RoboDK station: CuadrosElectricos.rdk

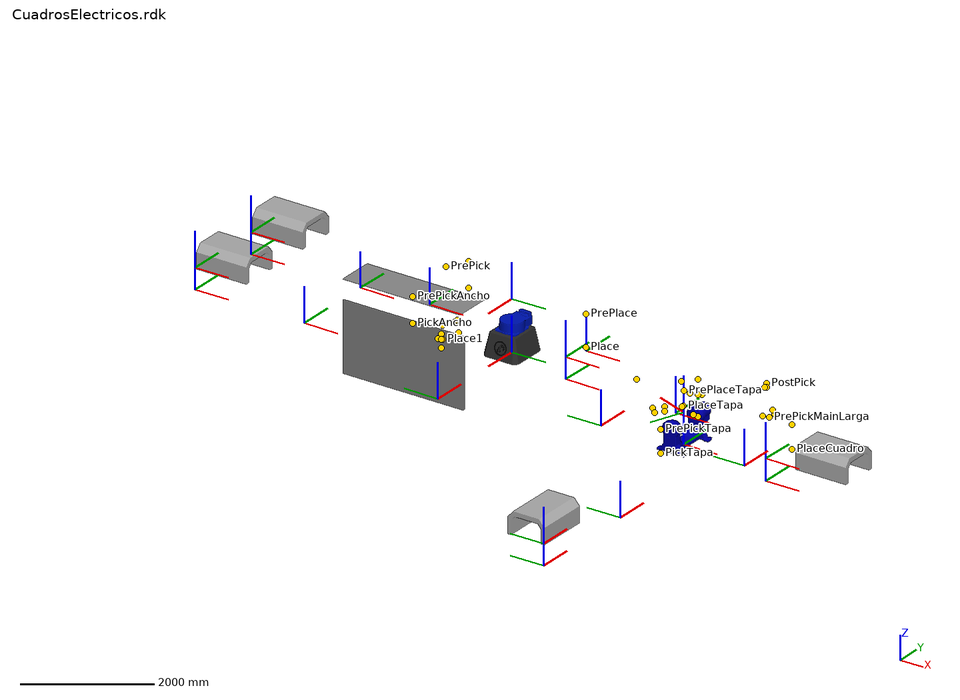
[picture v0: the station drawn from its stored meshes, robots at their saved joint values, targets as dots, program paths as lines]
Station CuadrosElectricos (saved by RoboDK 6.0.0). Poses are relative to the parent item; angles as X-Y-Z fixed-axis rotations.
Station parameters (name, value as stored): SensorCA, 0, SensorCL, 0, SensorCM, 0, SensorTapa, 0, SensorEtiqueta, 0, SensorFinalEtiqueta, 0, BendingHecho, 0, enCintaMain, 0, mesaOcupada, 0, LasDos, 0, planchaSoldada, 0, tapaPuesta, 0, EnCintaEtiquetar, 0, numero_planchaAncha, 0, numero_planchaLarga, 0, numero_planchaAncha1, 0, numero_planchaAncha2, 0, numero_planchaLarga1, 0, numero_planchaLarga2, 0, numero_planchaSoldada, 0, numero_tapaCuadro, 0, numero_cuadroConTapa, 0, numero_cuadroEtiquetada, 0, yaskawa_larga, 0, yaskawa_ancha, 0, abb_tapa, 0, parada_emergencia, 0
  - machining project Ajustes de mecanizado1: rotZ(0) | rotX(0)*rotY(0) | rotz(0) | onStart | onPathStart | onApproach | onPoint | onRetract | onFinish | SetRPM(%1) | SetTool(%1) | Extruder(%1) | default | default | OutOnMov(%1) | OutOffMov(%1) | onPathFinish | M_RunCode(%1)
  - folder Sistemas de Ref
    - frame World at (0, 0, 0) mm, rotated rx 0 ry 0 rz -90 deg
      - object Valla at (10, -2980, 0) mm, rotated rx 0 ry 0 rz 90 deg
      - object PedestalRobotPrensado at (0, 0, 0) mm, rotated rx 0 ry 0 rz 90 deg, size 633.4 x 700.2 x 375 mm, 1065353216 curves, geometry from Pedestal-H500mm-Type-2 (1).sld
      - object Suelo at (1170, 1000, -5) mm, size 11520 x 17280 x 0 mm, 1056816382 curves, geometry from PLUGIN_DISPLAY_DATAU
      - frame Frame_CintaCuadroInit at (300, 1190, 0) mm, rotated rx 0 ry 0 rz 90 deg
        - robot CintaCuadroIni: 1 axes
            modified DH rows (alpha deg, a mm, theta deg, d mm): 0, 0, 0, 0 linear
            base shift (0, 0, 0) mm, rotated rx 0 ry 90 rz 0 deg
            joint limits [-900000] to [900000]; home [0]; saved at [0]
          - frame FramePlanchaMain at (0, 0, 0) mm
      - frame Frame_CintaCuadroMid at (300, 3190, 0) mm, rotated rx 0 ry 0 rz 90 deg
        - robot CintaCuadroMid: 1 axes
            modified DH rows (alpha deg, a mm, theta deg, d mm): 0, 0, 0, 0 linear
            base shift (0, 0, 0) mm, rotated rx 0 ry 90 rz 0 deg
            joint limits [-900000] to [900000]; home [0]; saved at [0]
        - object SensorCM at (1880, 630, 370) mm, rotated rx 90 ry 0 rz -90 deg
      - frame Frame_CintaCuadroFinal at (1420, 5610, 0) mm, rotated rx 0 ry 0 rz 90 deg
        - robot CintaCuadroFini: 1 axes
            modified DH rows (alpha deg, a mm, theta deg, d mm): 0, 0, 0, 0 linear
            base shift (0, 0, 0) mm, rotated rx 0 ry 90 rz 0 deg
            joint limits [-900000] to [900000]; home [0]; saved at [0]
          - frame FrameEtiqueta at (0, 0, 0) mm
        - target CintaCuadroSoldadoIni (joint target) at (-550, 0, 366.5) mm; joints [3450] of CintaCuadroFini
        - target CintaCuadroSoldadoFin (joint target) at (2010, 0, 366.5) mm; joints [6010, -103.845, 100.785, 0, -114.63, -14.149, 0] of CintaCuadroFini
        - object tunelEtiqueta at (1000, 310, 760) mm, size 913.4 x 675.6 x 396.2 mm, geometry from tunel_andreu.stl
        - object SensorEtiqueta at (1240, 310, 690) mm, rotated rx 0 ry 90 rz 0 deg
        - object SensorFinalEtiqueta at (1880, 630, 370) mm, rotated rx 90 ry 0 rz -90 deg
      - frame Frame_CintaAnchoInit at (970, -5100, 0) mm, rotated rx 0 ry 0 rz 90 deg
        - robot CintaAnchoIni: 1 axes
            modified DH rows (alpha deg, a mm, theta deg, d mm): 0, 0, 0, 0 linear
            base shift (0, 0, 0) mm, rotated rx 0 ry 90 rz 0 deg
            joint limits [-900000] to [900000]; home [0]; saved at [0]
          - frame FramePlanchaAncha at (9, 0, 0) mm
        - object tunelAncha at (-2360, 3530, -20) mm, size 913.4 x 675.6 x 396.2 mm, geometry from tunel_andreu.stl
      - frame Frame_CintaAnchoFinal at (970, -3100, 0) mm, rotated rx 0 ry 0 rz 90 deg
        - robot Conveyor Belt Wide (2m): 1 axes
            modified DH rows (alpha deg, a mm, theta deg, d mm): 0, 0, 0, 0 linear
            base shift (0, 0, 0) mm, rotated rx 0 ry 90 rz 0 deg
            joint limits [-900000] to [900000]; home [0]; saved at [28.931]
        - object SensorCA at (1915, -40, 351.5) mm, rotated rx 90 ry 0 rz 90 deg
      - frame Frame_CintaLargoInit at (-490, -5100, 0) mm, rotated rx 0 ry 0 rz 90 deg
        - robot CintaLargoIni: 1 axes
            modified DH rows (alpha deg, a mm, theta deg, d mm): 0, 0, 0, 0 linear
            base shift (0, 0, 0) mm, rotated rx 0 ry 90 rz 0 deg
            joint limits [-900000] to [900000]; home [0]; saved at [0]
          - frame FramePlanchaLarga at (0, 0, 0) mm
        - object tunelLarga at (-2360, 3530, -20) mm, size 913.4 x 675.6 x 396.2 mm, geometry from tunel_andreu.stl
      - frame Frame_CintaLargoFinal at (-490, -3100, 0) mm, rotated rx 0 ry 0 rz 90 deg
        - robot Conveyor Belt Wide (2m): 1 axes
            modified DH rows (alpha deg, a mm, theta deg, d mm): 0, 0, 0, 0 linear
            base shift (0, 0, 0) mm, rotated rx 0 ry 90 rz 0 deg
            joint limits [-900000] to [900000]; home [0]; saved at [28.931]
        - object SensorCL at (1825, -40, 351.5) mm, rotated rx 90 ry 0 rz 90 deg
      - frame Frame_CintaTapaInit at (5690, 4560, 0) mm, rotated rx 0 ry 0 rz 180 deg
        - robot CintaTapaInit: 1 axes
            modified DH rows (alpha deg, a mm, theta deg, d mm): 0, 0, 0, 0 linear
            base shift (0, 0, 0) mm, rotated rx 0 ry 90 rz 0 deg
            joint limits [-900000] to [900000]; home [0]; saved at [0]
          - frame FrameTapa at (0, 0, 0) mm
        - object tunelTapa at (-2430, 3530, -20) mm, size 913.4 x 675.6 x 396.2 mm, geometry from tunel_andreu.stl
      - frame Frame_CintaTapaFinal at (3690, 4560, 0) mm, rotated rx 0 ry 0 rz 180 deg
        - robot CintaTapaFinal: 1 axes
            modified DH rows (alpha deg, a mm, theta deg, d mm): 0, 0, 0, 0 linear
            base shift (0, 0, 0) mm, rotated rx 0 ry 90 rz 0 deg
            joint limits [-900000] to [900000]; home [0]; saved at [3450]
        - object SensorTapa at (1710, 620, 355) mm, rotated rx 90 ry 0 rz -90 deg
    - frame RobotPrensado at (0, 0, 880) mm, rotated rx 0 ry 0 rz -90 deg
      - robot Yaskawa MH24 Prensado (model Yaskawa MH24): 6 axes, payload 24 kg, reach 1730 mm, repeatability 0.06 mm, weight 268 kg
          modified DH rows (alpha deg, a mm, theta deg, d mm): 0, 0, 0, 505; -90, 150, -90, 0; 0, 760, 0, 0; -90, 200, 0, 795; 90, 0, 0, 0; -90, 0, 0, 100
          base shift (0, 0, -505) mm
          joint limits [-180, -105, -170, -200, -150, -455] to [180, 155, 240, 200, 150, 455]; home [0, 0, 0, 0, 0, 0]; saved at [-120.522, 54.399, 24.171, 0, -59.772, 120.522]
        - tool EPick Bend, TCP at (0, 0, 185) mm
    - frame RobotPaletizado at (5060, -1180, 0) mm, rotated rx 0 ry 0 rz 90 deg
      - robot ABB Paletizado (model ABB IRB 1660-4/1.55): 6 axes, payload 4 kg, reach 1550 mm, repeatability 0.02 mm, weight 257 kg
          modified DH rows (alpha deg, a mm, theta deg, d mm): 0, 0, 0, 481.5; -90, 150, -90, 0; 0, 700, 0, 0; -90, 110, 0, 678; 90, 0, 0, 0; -90, 0, 180, 135
          joint limits [-180, -90, -238, -175, -120, -400] to [180, 150, 79, 175, 120, 400]; home [0, 0, 0, 0, 0, 0]; saved at [16.288, 32.625, 48.175, 16.099, -82.213, 87.26]
        - tool EPick Gripper, TCP at (0, 30, 180) mm
      - frame Cinta_Mesa at (0, 0, 0) mm
        - target PrePickMainLarga (Cartesian target) at (777.3, 95, 463.61) mm, rotated rx 88.94 ry 0.2 rz 90.34 deg; joints [11.364, 25.315, 71.994, 11.14, -98.231, 91.211, 0] of ABB Paletizado
        - target PickMainLarga (Cartesian target) at (927.3, 95, 463.61) mm, rotated rx 88.94 ry 0.2 rz 90.33 deg; joints [8.631, 27.949, 59.348, 8.295, -88.383, 89.412, 0] of ABB Paletizado
        - target PrePickMainAncha (Cartesian target) at (777, 210.74, 455.18) mm, rotated rx 88.94 ry 0.2 rz 90.34 deg; joints [24.29, 27.02, 68.896, 24.11, -96.462, 92.216, 0] of ABB Paletizado
        - target PickMainAncha (Cartesian target) at (1028.89, 210.74, 455.18) mm, rotated rx 88.94 ry 0.2 rz 90.34 deg; joints [16.288, 32.625, 48.175, 16.099, -82.213, 87.26, 0] of ABB Paletizado
        - target PostPick (Cartesian target) at (758.49, 121.16, 1025.46) mm, rotated rx 88.94 ry 0.2 rz 90.34 deg; joints [15.024, -32.079, 48.401, 41.2, -22.631, 50.585, 0] of ABB Paletizado
        - target Giro180_P (Cartesian target) at (758, 121, 965.48) mm, rotated rx -88.95 ry -1.49 rz -89.69 deg; joints [15.162, -32.222, 48.464, 41.609, -22.656, 228.889, 0] of ABB Paletizado
        - target PrePlaceMain (Cartesian target) at (-1.33, 767.63, 965.52) mm, rotated rx -88.95 ry -1.51 rz -8.65 deg; joints [96.19, -32.22, 48.46, 41.6, -22.65, 228.88, 0] of ABB Paletizado
        - target PlaceMainLarga (Cartesian target) at (82, 907.5, 524) mm, rotated rx -90 ry 0 rz 0 deg; joints [82.121, 11.477, 61.016, -8.257, -72.663, -87.524, 0] of ABB Paletizado
        - target PlaceMainAncha (Cartesian target) at (100, 995, 525) mm, rotated rx -90 ry 0 rz 0 deg; joints [81.634, 16.501, 53.189, -8.912, -69.916, -86.918, 0] of ABB Paletizado
      - target Inicio (Cartesian target) at (790.15, 181.03, 936.03) mm, rotated rx 88.94 ry 0.2 rz 90.33 deg; joints [20.625, -24.78, 52.397, 37.542, -34.674, 57.118, 0] of ABB Paletizado
      - target PrePickTapa (Cartesian target) at (-1018.21, 818.52, 780.95) mm, rotated rx -179.33 ry -0.3 rz -86.99 deg; joints [140.371, 40.682, -38.487, -0.236, 88.496, 47.366, 0] of ABB Paletizado
      - target PickTapa (Cartesian target) at (-1018.21, 818.52, 380.95) mm, rotated rx -179.33 ry -0.3 rz -86.99 deg; joints [140.371, 46.29, -14.025, -0.277, 58.427, 47.505, 0] of ABB Paletizado
      - target PrePlaceTapa (Cartesian target) at (77.73, 1160.64, 889) mm, rotated rx -179.72 ry 0.67 rz -177.45 deg; joints [86.193, 25.731, -24.216, -0.695, 88.694, 83.664, 0] of ABB Paletizado
      - target PrePlaceTapaG1 (Cartesian target) at (239.54, 1017.6, 1052.03) mm, rotated rx 108.26 ry -87.33 rz -106.91 deg; joints [60.84, 25.81, -11.886, 81.018, 119.265, 70.969, 0] of ABB Paletizado
      - target PrePlaceTapaG2 (Cartesian target) at (239.54, 1017.6, 802.03) mm, rotated rx 108.26 ry -87.33 rz -106.91 deg; joints [60.84, 30.993, 1.938, 71.52, 114.698, 50.23, 0] of ABB Paletizado
      - target PrePlaceTapaG3 (Cartesian target) at (243.81, 1163, 773.67) mm, rotated rx 105.66 ry -86.91 rz -104.31 deg; joints [63.869, 42.236, -14.07, 75.44, 113.553, 55.604, 0] of ABB Paletizado
      - target PlaceTapa (Cartesian target) at (86.58, 1170.89, 626.96) mm, rotated rx -179.79 ry -0.03 rz -176.92 deg; joints [85.58, 27.86, -5.32, 0, 67.67, 82.5, 0] of ABB Paletizado
      - target PrePickCuadro (Cartesian target) at (51.62, 1181.79, 1052.12) mm, rotated rx -179.77 ry 0.7 rz 177.71 deg; joints [87.684, 33.633, -50.583, -0.729, 107.181, 89.762, 0] of ABB Paletizado
      - target PickCuadro (Cartesian target) at (56.65, 1179.89, 632.15) mm, rotated rx -179.77 ry 0.7 rz 177.71 deg; joints [87.43, 28.34, -6.48, -0.75, 68.37, 90, 0] of ABB Paletizado
      - target PrePlaceCuadro (Cartesian target) at (82.65, -808.13, 869.56) mm, rotated rx 179.56 ry -0.46 rz -2.19 deg; joints [-84.012, -4.668, 13.456, 0.401, 80.709, 98.117, 0] of ABB Paletizado
      - target PlaceCuadro (Cartesian target) at (82.65, -808.13, 469.56) mm, rotated rx 179.56 ry -0.46 rz -2.19 deg; joints [-84.012, 5.511, 38.703, 0.556, 45.284, 97.79, 0] of ABB Paletizado
    - frame RobotSoldador at (2530, -1300, 0) mm, rotated rx 0 ry 0 rz 90 deg
      - robot ABB Soldador (model ABB IRB 1660-4/1.55): 6 axes, payload 4 kg, reach 1550 mm, repeatability 0.02 mm, weight 257 kg
          modified DH rows (alpha deg, a mm, theta deg, d mm): 0, 0, 0, 481.5; -90, 150, -90, 0; 0, 700, 0, 0; -90, 110, 0, 678; 90, 0, 0, 0; -90, 0, 180, 135
          joint limits [-180, -90, -238, -175, -120, -400] to [180, 150, 79, 175, 120, 400]; home [0, 0, 0, 0, 0, 0]; saved at [36.59, -2.68, -230.3, -70.7, 119.79, -124.86]
        - tool Welding Gun, TCP at (86, 0, 451.5) mm, rotated rx 0 ry 36 rz 0 deg
      - target Inicio_Soldador (Cartesian target) at (200.82, -506.97, 837.81) mm, rotated rx 94.58 ry 80.61 rz 52.68 deg; joints [36.59, -2.68, -230.3, -70.7, 119.79, -124.86, 0] of ABB Soldador
      - target prePIS (Cartesian target) at (-101.3, -1007.69, 623.69) mm, rotated rx 134.47 ry 88.84 rz 90.8 deg; joints [53.05, -51.812, -173.339, -59.361, 109.58, -131.05, 0] of ABB Soldador
      - target PIS (Cartesian target) at (36.12, -1138.87, 621.01) mm, rotated rx 134.47 ry 88.84 rz 90.8 deg; joints [65.969, -54.136, -168.246, -51.218, 100.348, -134.197, 0] of ABB Soldador
      - target PFS (Cartesian target) at (36.09, -1137.26, 541.02) mm, rotated rx 134.47 ry 88.84 rz 90.8 deg; joints [65.922, -59.336, -166.814, -51.849, 102.718, -137.187, 0] of ABB Soldador
      - target postPFS (Cartesian target) at (-72.39, -1033.69, 543.14) mm, rotated rx 134.47 ry 88.84 rz 90.8 deg; joints [55.809, -57.49, -171.254, -58.794, 109.811, -135.353, 0] of ABB Soldador
    - frame Pick at (-1500, 0, 370) mm
      - target PrePick (Cartesian target) at (160, 190, 600) mm, rotated rx -180 ry 0 rz -90 deg; joints [-98.253, 31.893, -1.848, 0, -56.259, 98.253, 0] of Yaskawa MH24 Prensado
      - target PrePickAncho (Cartesian target) at (160, -670, 440) mm, rotated rx -180 ry 0 rz -90 deg; joints [-63.435, 49.441, 15.409, 180, 55.968, -116.565, 0] of Yaskawa MH24 Prensado
      - target PrePickLargo (Cartesian target) at (160, 790, 440) mm, rotated rx -180 ry 0 rz -90 deg; joints [-120.522, 54.399, 24.171, 0, -59.772, 120.522, 0] of Yaskawa MH24 Prensado
      - target PickAncho (Cartesian target) at (160, -670, 0) mm, rotated rx -180 ry 0 rz -90 deg; joints [-63.435, 68.099, 15.642, 180, 37.543, -116.565, 0] of Yaskawa MH24 Prensado
      - target PickLargo (Cartesian target) at (160, 790, 0) mm, rotated rx -180 ry 0 rz -90 deg; joints [-120.522, 72.326, 24.429, 180, 42.104, -59.478, 0] of Yaskawa MH24 Prensado
    - frame Place at (1350, 0, 400) mm
      - target PrePlace (Cartesian target) at (0, 0, 610) mm, rotated rx -180 ry 0 rz 90 deg; joints [90, 30.642, -0.787, 0, -58.571, 90, 0] of Yaskawa MH24 Prensado
      - target Place (Cartesian target) at (0, 0, 56) mm, rotated rx 180 ry 0 rz 90 deg; joints [90, 53.307, -7.669, -180, 29.024, 270, 0] of Yaskawa MH24 Prensado
    - frame MesaGiratoria at (3900, -1100, 0) mm
      - robot Yaskawa Giratoria (model Motoman MOTOPOS-D250F): 2 axes
          modified DH rows (alpha deg, a mm, theta deg, d mm): 0, 0, 0, 0; 90, 0, 0, 0
          base shift (0, 0, 380) mm, rotated rx -90 ry 0 rz 0 deg
          joint limits [-135, -200] to [135, 200]; home [0, 0]; saved at [0, -200]
        - frame Engranaje at (0, 0, 0) mm
      - target Inici (Cartesian target) at (0, 0, 530) mm, rotated rx 0 ry 0 rz 160 deg; joints [0, -200, -7.748, -180, 29.277, 270, 0] of Yaskawa Giratoria
      - target Giro90 (joint target) at (0, 0, 530) mm, rotated rx 0 ry 0 rz -110 deg; joints [0, -110, 19.031, 0, -41.803, 121.092, 0] of Yaskawa Giratoria
      - target Esquina0 (Cartesian target) at (0, 0, 530) mm, rotated rx 0 ry 0 rz -20 deg; joints [0, -20, 0, 0, 0, 0, 0] of Yaskawa Giratoria
      - target Esquina1 (Cartesian target) at (0, 0, 530) mm, rotated rx 0 ry 0 rz 47.5 deg; joints [0, 47.5, 0, 0, 0, 0, 0] of Yaskawa Giratoria
      - target Esquina2 (Cartesian target) at (0, 0, 530) mm, rotated rx 0 ry 0 rz 160 deg; joints [0, 160, 0, 0, 0, 0, 0] of Yaskawa Giratoria
      - target Esquina3 (Cartesian target) at (0, 0, 530) mm, rotated rx 0 ry 0 rz -175 deg; joints [0, 185, 0, 0, 0, 0, 0] of Yaskawa Giratoria
      - target Final (Cartesian target) at (0, 0, 530) mm, rotated rx 0 ry 0 rz 180 deg; joints [0, 180, -7.748, -180, 29.277, 270, 0] of Yaskawa Giratoria
    - frame Bending at (0, -1940, 0) mm, rotated rx 0 ry 0 rz 90 deg
      - object tapa_prensa at (-450, 120, 1965) mm, size 640 x 2140 x 5 mm, geometry from tapa_prensa3.stl
      - object tapa_darrere at (-725, 110, 990) mm, rotated rx 0 ry 0 rz 90 deg, size 2197.8 x 29.7 x 1217.7 mm, 1064168942 curves, geometry from tapaor3.stl
      - robot Press Brake: 1 axes
          modified DH rows (alpha deg, a mm, theta deg, d mm): 0, 0, 0, 0 linear
          joint limits [0] to [230]; home [0]; saved at [0]
      - target Home (Cartesian target) at (557.12, 0, 874.46) mm, rotated rx -177.4 ry 0 rz -90 deg; joints [0, 37.6, 0, 0, -55, 90, 0] of Yaskawa MH24 Prensado
      - target Place1 (joint target) at (144.16, 0, 929.49) mm, rotated rx 0 ry -31.66 rz 0 deg; joints [0, 79.41, 41.34, 0, 96.41, 0, 0] of Yaskawa MH24 Prensado
      - target Place2 (joint target) at (144.16, 0, 929.49) mm, rotated rx 0 ry 31.66 rz -180 deg; joints [0, 79.41, 41.34, 0, 96.41, 180, 0] of Yaskawa MH24 Prensado
      - target BajaPrensa1 (joint target) at (144.16, 0, 929.49) mm, rotated rx 0 ry -31.66 rz 0 deg; joints [0, 79.41, 41.34, 0, 96.41, 0, 230] of Yaskawa MH24 Prensado
      - target BajaPrensa2 (joint target) at (144.16, 0, 1159.49) mm, rotated rx 0 ry 31.66 rz -180 deg; joints [0, 79.41, 41.34, 0, 96.41, 180, 230] of Yaskawa MH24 Prensado
      - target Bend1 (joint target) at (101.51, 0, 1035) mm, rotated rx 0 ry -60 rz 0 deg; joints [0, 64.383, 27.581, 0, 66.801, 0, 230] of Yaskawa MH24 Prensado
      - target BendA1 (joint target) at (57.18, 30, 968.22) mm, rotated rx 0 ry -60 rz 0 deg; joints [0, 71.944, 37.304, 0, 64.64, 0, 230] of Yaskawa MH24 Prensado
      - target Bend2 (joint target) at (101.52, 0, 1035.05) mm, rotated rx 0 ry 60 rz -180 deg; joints [0, 64.38, 27.58, 0, 66.8, 180, 230] of Yaskawa MH24 Prensado
      - target BendA2 (joint target) at (65.36, -30, 970.72) mm, rotated rx 0 ry 60 rz -180 deg; joints [0, 70.932, 35.526, 0, 65.405, 180, 230] of Yaskawa MH24 Prensado
      - target AbrePrensa1 (joint target) at (101.51, 0, 805) mm, rotated rx 0 ry -60.01 rz 0 deg; joints [0, 64.378, 27.576, 0, 66.792, 0, 0] of Yaskawa MH24 Prensado
      - target AbrePrensa2 (joint target) at (101.49, 0, 805) mm, rotated rx 0 ry 60.01 rz -180 deg; joints [0, 64.38, 27.58, 0, 66.79, 180, 0] of Yaskawa MH24 Prensado
      - target Retract1 (Cartesian target) at (485.32, 30, 1066.8) mm, rotated rx -180 ry -87.45 rz 180 deg; joints [0, 27.86, -21.47, 0, 46.78, 0, 0] of Yaskawa MH24 Prensado
      - target Retract2 (Cartesian target) at (488.99, -30, 1096.85) mm, rotated rx -180 ry 87.44 rz 0 deg; joints [0, 26.34, -21.22, 0, 45, -180, 0] of Yaskawa MH24 Prensado
      - target Gir180 (Cartesian target) at (482.67, -30, 1126.45) mm, rotated rx 180 ry 87.43 rz 0 deg; joints [0, 25.54, -19.95, 0, 42.92, 180, 0] of Yaskawa MH24 Prensado
  - folder Plantillas Objetos
    - object plantilla_planchaLarga at (-4880, 800, 371.5) mm, size 323.4 x 693 x 2.3 mm, geometry from planxa1.3.stl
    - object plantilla_planchaLarga1 at (-30, -1838.49, 1035) mm, rotated rx -60 ry 0 rz 180 deg, size 317 x 589.8 x 91.7 mm, geometry from planxa2.2_intermig.stl
    - object plantilla_planchaLarga2 at (30, -1839.49, 1035) mm, rotated rx -60 ry 0 rz 180 deg, size 316.6 x 499.9 x 91.6 mm, geometry from planxa2.2.stl
    - object plantilla_planchaAncha at (-4831, -665, 371.5) mm, rotated rx 0 ry 0 rz 90 deg
    - object plantilla_planchaAncha1 at (-30, -1888.49, 965) mm, rotated rx 0 ry 60 rz -90 deg
    - object plantilla_planchaAncha2 at (30, -1888.49, 965) mm, rotated rx 0 ry -60 rz 90 deg
    - object plantilla_tapaCuadro at (4250, -5420, 366.5) mm
    - object plantilla_planchaSoldada at (3900, -1100, 530) mm, rotated rx 0 ry 0 rz -90 deg
    - object plantilla_cuadroConTapa at (3900, -1100, 530) mm, rotated rx 0 ry 0 rz -90 deg
    - object plantilla_etiqueta at (6500, -1070, 465) mm, rotated rx 0 ry 0 rz 90 deg, size 225.7 x 166.7 x 1.6 mm, geometry from etiqueta.stl
  - folder Programas
    - Python program reset (listed below)
    - Python program main (listed below)

--- Python program reset ---
"""Este módulo ayuda al reseteo de la estación.

Establece parámetros a 0, devuelve las cintas a su
posición original y elimina objetos."""

from robodk import robolink, robomath
from modulos_python import simulation as sim, variables as var
import json

def reset_cinta(mecanismos : list[str]):
    """Devuelve la cinta a la posición 0 y valida que exista el mecanismo."""
    RDK = robolink.Robolink()

    for nombre_cinta in mecanismos:
        item_cinta = RDK.Item(nombre_cinta, robolink.ITEM_TYPE_ROBOT)
        if not item_cinta.Valid():
            raise RuntimeError(RDK.ShowMessage(f"Cinta: {nombre_cinta} no existe, revisa nombres"))

        if item_cinta.Name() == var.mesa_giratoria:
            target_ini_mesa = RDK.Item("Inici", robolink.ITEM_TYPE_TARGET)

            if not target_ini_mesa.Valid():
                raise RuntimeError("Target de esquina inválido. Revisa nombres")

            item_cinta.MoveJ(target_ini_mesa)
            continue
        item_cinta.setJoints(robomath.Mat([[0]]))

def reset_param():
    """Carga los parámetros del JSON persistente y los reinicia a 0."""

    if not var.JSON_PARAM_PATH.exists():
        return
    with var.JSON_PARAM_PATH.open("r", encoding="utf-8") as f:
        data = json.load(f)

    parametros = data.get("parametros", []) if isinstance(data, dict) else data
    for nombre in parametros:
        sim.setDO(str(nombre), 0)

def eliminar_duplicados(frame_name : str):
    RDK = robolink.Robolink()

    frame = RDK.Item(frame_name, robolink.ITEM_TYPE_FRAME)
    if not frame.Valid():
            raise RuntimeError(RDK.ShowMessage(f"Frame: {frame_name} no existe, revisa nombres"))

    lista_objetos = frame.Childs()

    if not lista_objetos:
        return

    for idx in lista_objetos:
        idx.Delete()

eliminar_duplicados("FramePlanchaAncha")
eliminar_duplicados("FramePlanchaLarga")
eliminar_duplicados("FramePlanchaMain")
eliminar_duplicados("FrameTapa")
eliminar_duplicados("FrameEtiqueta")
eliminar_duplicados("Engranaje")

reset_param()
reset_cinta(var.mecanismos)

--- Python program main ---
"""Archivo principal que ejecuta todas las acciones de los distintos módulos.

Se caracteriza por el uso de hilos para cada acción o conjunto de acciones
necesarias para la automatización de cuadros eléctricos.

El uso de hilos permite ejecutar instancias en paralelo, por ejemplo mover
cintas o coordinar robots simultáneamente."""

from modulos_python.entorno import preparar_entorno
preparar_entorno()

from modulos_python import bending, sensor, soldar, variables, mqtt, bbdd
from modulos_python import mover_cinta as mc, pick_place as pp, simulation as sim

from robodk import robolink
import threading
import time

mqtt.conectar()
#bbdd.conectar()

sim.setDO("yaskawa_larga", 1)
sim.setDO("yaskawa_ancha", 1)
sim.setDO("abb_tapa", 1)

def _thread_excepthook(args):
    """Se hace uso de este método interno para imprimir por pantalla los errores que
    surjan en tiempo de ejecución, es muy útil porque nos dice en que hilo ha fallado
    y devuelve el mensaje que elevan las excepciones en las funciones internas al hilo."""

    RDK = robolink.Robolink()

    RDK.ShowMessage(f"[ThreadError] {args.thread.name}: {args.exc_type.__name__}: {args.exc_value}")

threading.excepthook = _thread_excepthook

# Los siguientes hilos mueven las cintas por donde llegan los objetos.
def hilo_cinta_larga():
    """Hilo que mueve la cinta de planchas largas."""
    while True:
        sim.waitDI("yaskawa_larga" , 1)
        mc.mover_cinta_larga()
        time.sleep(0.01)

def hilo_cinta_ancha():
    """Hilo que mueve la cinta de planchas anchas."""
    while True:
        sim.waitDI("yaskawa_ancha" , 1)
        mc.mover_cinta_ancha()
        time.sleep(0.01)

def hilo_cinta_tapa():
    """Hilo que mueve la cinta de tapas."""
    while True:
        sim.waitDI("abb_tapa" , 1)
        mc.mover_cinta_tapa()
        time.sleep(0.01)

def hilo_cinta_main():
    """Hilo que mueve la cinta principal cuando hay pieza disponible."""
    while True:
        mc.mover_cinta_main()
        time.sleep(0.01)

def hilo_cinta_etiquetado():
    """Hilo que mueve la cinta final de etiquetado."""
    while True:
        mc.mover_cinta_cuadro_acabada()
        time.sleep(0.01)

# Los siguientes hilos llaman a funciones donde los robots realizan movimientos de pick & place, prensado y soldado
def hilo_yaskawa():
    """Este hilo llama a la secuencia de movimientos pick->bending->place
    de un tipo de planchas o otro. Para no depender de la salida digital
    que se genera el objeto, se implemento una cola para cada sensor donde
    se guarda el objeto una vez el sensor detecte que hay un objeto.
    Así la información es más persistente en tiempo de ejecución."""

    cola_ancha = variables.objetos_pendientes["SensorCA"]
    cola_larga = variables.objetos_pendientes["SensorCL"]

    while True:

        nombre_larga = cola_larga.get()
        pp.pick_plancha_larga(nombre_larga)
        bending.bending_plancha_larga(nombre_larga)
        pp.place_cinta_main()
        variables.alternancia.put("larga")

        nombre_ancha = cola_ancha.get()
        pp.pick_plancha_ancha(nombre_ancha)
        bending.bending_plancha_ancha(nombre_ancha)
        pp.place_cinta_main()
        variables.alternancia.put("ancha")

        time.sleep(0.01)

def hilo_abb_paletizado():
    """Hilo del abb paletizado que decide que tarea hace primero segun la logica de la automatización."""

    RDK = robolink.Robolink()

    while True:
        if RDK.getParam("tapaPuesta") == 1 and not variables.cola_cuadrosTapa.empty():
            pp.place_cuadro_acabada()
        elif RDK.getParam("planchaSoldada") == 1 and not variables.objetos_pendientes["SensorTapa"].empty():
            pp.place_tapa_en_mesa()
        elif RDK.getParam("mesaOcupada") == 0 and not variables.objetos_pendientes["SensorCM"].empty():
            pp.place_plancha_mesa()
        else:
            time.sleep(0.01)

def hilo_abb_soldador():
    """Hilo que ejecuta la secuencia de soldadura."""
    while True:
        soldar.iniciar()
        time.sleep(0.01)

# Hilos de sensores para detectar objetos en cada cinta.
def hilo_sensorCA():
    """Hilo del sensor de planchas anchas."""
    sensor.detectar_objeto("SensorCA", "FramePlanchaAncha")

def hilo_sensorCL():
    """Hilo del sensor de planchas largas."""
    sensor.detectar_objeto("SensorCL", "FramePlanchaLarga")

def hilo_sensorCM():
    """Hilo del sensor de la cinta principal."""
    sensor.detectar_objeto("SensorCM", "FramePlanchaMain")

def hilo_sensorTapa():
    """Hilo del sensor de tapas."""
    sensor.detectar_objeto("SensorTapa", "FrameTapa")

def hilo_sensorEtiqueta():
    """Hilo del sensor de la cinta de etiquetado."""
    sensor.detectar_objeto("SensorEtiqueta", "FrameEtiqueta")

def hilo_sensorFinalEtiqueta():
    """Hilo del sensor de la cinta de etiquetado."""
    sensor.detectar_objeto("SensorFinalEtiqueta", "FrameEtiqueta")

""" Lista para guardar todos los hilos que se van a ejecutar
en la estación, el parametro name se usa darle cuando
ocurra un error, que se imprima por mensaje el nombre del hilo."""
threads = [
    threading.Thread(target=hilo_cinta_larga, name="cinta_larga"),
    threading.Thread(target=hilo_cinta_ancha, name="cinta_ancha"),
    threading.Thread(target=hilo_cinta_main, name="cinta_main"),
    threading.Thread(target=hilo_cinta_tapa, name="cinta_tapa"),
    threading.Thread(target=hilo_cinta_etiquetado, name="cinta_etiquetado"),

    threading.Thread(target=hilo_yaskawa, name="yaskawa"),
    threading.Thread(target=hilo_abb_paletizado, name="paletizado"),
    threading.Thread(target=hilo_abb_soldador, name="soldador"),

    threading.Thread(target=hilo_sensorCA, name="sensor_ca"),
    threading.Thread(target=hilo_sensorCL, name="sensor_cl"),
    threading.Thread(target=hilo_sensorCM, name="sensor_cm"),
    threading.Thread(target=hilo_sensorTapa, name="sensor_tapa"),
    threading.Thread(target=hilo_sensorEtiqueta, name="sensor_etiqueta"),
    threading.Thread(target=hilo_sensorFinalEtiqueta, name="sensor_final_etiqueta")
]

# Se inicializan todos los hilos a la vez
for t in threads:
    t.start()
